{attribute 'qualified_only'}
VAR_GLOBAL
	bLedLight		AT %Q* :BOOL;			//カメラ用LED照明
END_VAR

(* stored: Version 1.1.0.1, ProductVersion 3.1.4024.12
   GVL GVL_Vision: Id {19ce6139-658e-4644-9138-c7378a7b0ab0} *)
